TYPE "TrkMng_Move"
VERSION : 0.1
// Block: TrkMng_Move
   STRUCT
      SelButton : Bool;
      PasteButton : Bool;
      DeleteButton : Bool;
      InfoButton : Bool;
      PasteButton_Visibile : Bool;
      DeleteButton_Visibile : Bool;
      SelectButton_Visibile : Bool;
      SelectButton_Selected : Bool;
   END_STRUCT;

END_TYPE
